// TIA Portal V18 export
TYPE "CheckOut_ShW"
// stored: IsFailsafeCompliant false
   STRUCT
      Trigger : Bool;
      SubStationResult : Int;
      NGCode : DInt;
      S_MainID : String[120];
      S_CarrierID : Int;
      S_CompletedProductID : String[48];
      S_PackageBatchID : String[48];
      Result : Int;
      Completed : Bool;
      S_ComponentID { S7_SetPoint := 'True'} : "ComponentID_ShW";
      S_BatchID { S7_SetPoint := 'True'} : "batchID_ShW";
      S_SubAssemblyID : "SubAssemblyID_ShW";
      S_OperatorNo : Struct
         _1 : String[48];
         _2 : String[48];
         _3 : String[48];
         _4 : String[48];
         _5 : String[48];
      END_STRUCT;
   END_STRUCT;
END_TYPE
